ABB RAPID module: RobData.mod

MODULE RobData
    PERS num nHeigh:=-2.5;
	CONST speeddata vSlow:=[10,5,5,1000];
	CONST robtarget pTemp:=[[36.61,-311.94,82.16],[3.72224E-05,-1,-4.64438E-05,2.60135E-05],[-1,-1,-1,0],[9E+09,9E+09,9E+09,9E+09,9E+09,9E+09]];
	CONST speeddata vSlowA:=[2,5,5,1000];
    PERS robtarget phome1:=[[-40.4314,-257.966,143.781],[4.99019E-05,-0.667497,0.744613,6.30517E-05],[-2,-1,-1,0],[9E+09,9E+09,9E+09,9E+09,9E+09,9E+09]];
    PERS robtarget phome:=[[-122.06,-373,117.55],[3.74264E-05,-0.659781,0.751458,3.53401E-05],[-2,-1,-1,0],[9E+09,9E+09,9E+09,9E+09,9E+09,9E+09]];
	PERS robtarget pPickWait:=[[-121.80,-372.62,142.89],[4.48442E-05,-0.659779,0.751459,4.07139E-05],[-2,-1,-1,0],[9E+09,9E+09,9E+09,9E+09,9E+09,9E+09]];
    PERS robtarget pTCPCalib:=[[38.86,-315.26,82.1995],[4.51814E-05,-6.4519E-06,-1,-4.06358E-05],[-1,-1,-1,0],[9E+09,9E+09,9E+09,9E+09,9E+09,9E+09]];

    PERS robtarget pPass1:=[[200.53,-307.58,242.84],[0.299987,0.731588,0.298484,-0.534504],[-1,-1,-1,0],[9E+09,9E+09,9E+09,9E+09,9E+09,9E+09]];
    PERS robtarget pPass2:=[[887.04,835.36,1127.78],[0.0262232,0.74592,-0.665204,-0.0204732],[0,-2,-1,0],[9E+09,9E+09,9E+09,9E+09,9E+09,9E+09]];
    PERS robtarget pAssembly:=[[0,0,118],[0,-1,0,0],[-1,0,-1,0],[9E+09,9E+09,9E+09,9E+09,9E+09,9E+09]];
	PERS robtarget pAssem:=[[354.53,109.44,1307.28],[0.522631,-0.494622,0.5135,0.467465],[0,-1,-1,0],[9E+09,9E+09,9E+09,9E+09,9E+09,9E+09]];
    PERS robtarget pAssBase:=[[225.06,-308.31,118.65],[0.0102026,-0.99364,-0.111268,-0.0139692],[-1,0,-1,0],[9E+09,9E+09,9E+09,9E+09,9E+09,9E+09]];
    PERS robtarget pCali2Temp:=[[221.471,-305.943,140.42],[3.87751E-06,0.113366,-0.993553,-6.74824E-05],[-1,0,-1,0],[9E+09,9E+09,9E+09,9E+09,9E+09,9E+09]];
    VAR robtarget pActPos:=[[752.23,113.39,1307.28],[0.522626,-0.494634,0.513503,0.467454],[0,-2,0,0],[9E+09,9E+09,9E+09,9E+09,9E+09,9E+09]];
    PERS tooldata tGripper:=[TRUE,[[0,0,108],[0,0,0,-1]],[1,[0,0,0.001],[1,0,0,0],0,0,0]];
    PERS tooldata tcp1:=[TRUE,[[-134.881,-2.6021,210.993],[0.472574,-0.509839,-0.505206,0.511376]],[0.001,[0,0,0.001],[1,0,0,0],0,0,0]];
    PERS tooldata tcp2:=[TRUE,[[-134.881,-2.6021,210.993],[0.472574,-0.509839,-0.505206,0.511376]],[0.001,[0,0,0.001],[1,0,0,0],0,0,0]];
    PERS tooldata tCurTool:=[TRUE,[[0.0931091,-0.0380325,108],[0.998678,-1.1568E-12,-2.18595E-12,-0.0514118]],[1,[0,0,0.001],[1,0,0,0],0,0,0]];
    PERS wobjdata AssFrame:=[FALSE,TRUE,"",[[227.126,-306.421,7],[0.49417,0,0,-0.869366]],[[0,0,0],[1,0,0,0]]];
    PERS pose posRel:=[[27.92,-310.994,91.58],[3.54519E-05,-0.70071,-0.713446,3.18553E-08]];
    !the position of insert action
    PERS robtarget pccd2Calib{9}:=[[[221.89,-312.11,153.7],[6.08179E-05,-0.667482,0.744626,7.205E-05],[-1,0,0,0],[9E+09,9E+09,9E+09,9E+09,9E+09,9E+09]],[[221.89,-308.11,153.7],[6.08179E-05,-0.667482,0.744626,7.205E-05],[-1,0,0,0],[9E+09,9E+09,9E+09,9E+09,9E+09,9E+09]],[[221.89,-304.11,153.7],[6.08179E-05,-0.667482,0.744626,7.205E-05],[-1,0,0,0],[9E+09,9E+09,9E+09,9E+09,9E+09,9E+09]],[[225.89,-312.11,153.7],[6.08179E-05,-0.667482,0.744626,7.205E-05],[-1,0,0,0],[9E+09,9E+09,9E+09,9E+09,9E+09,9E+09]],[[225.89,-308.11,153.7],[6.08179E-05,-0.667482,0.744626,7.205E-05],[-1,0,0,0],[9E+09,9E+09,9E+09,9E+09,9E+09,9E+09]],[[225.89,-304.11,153.7],[6.08179E-05,-0.667482,0.744626,7.205E-05],[-1,0,0,0],[9E+09,9E+09,9E+09,9E+09,9E+09,9E+09]],[[229.89,-312.11,153.7],[6.08179E-05,-0.667482,0.744626,7.205E-05],[-1,0,0,0],[9E+09,9E+09,9E+09,9E+09,9E+09,9E+09]],[[229.89,-308.11,153.7],[6.08179E-05,-0.667482,0.744626,7.205E-05],[-1,0,0,0],[9E+09,9E+09,9E+09,9E+09,9E+09,9E+09]],[[229.89,-304.11,153.7],[6.08179E-05,-0.667482,0.744626,7.205E-05],[-1,0,0,0],[9E+09,9E+09,9E+09,9E+09,9E+09,9E+09]]];
    PERS string sCCD;
    PERS string sFirstStr;
    PERS string sSecondStr;
    PERS num Zangle:=-96.2517;
    PERS num Yangle:=0.00908074;
    PERS num Xangle:=179.998;
    VAR string CCD1X{9}:=["","","","","","","","",""];
    VAR string CCD1Y{9}:=["","","","","","","","",""];
    VAR string CCD2X{9}:=["","","","","","","","",""];
    VAR string CCD2Y{9}:=["","","","","","","","",""];
    PERS NUM ARRAY{9}:=[3,6,9,8,5,2,1,4,7];
    VAR string sCCD1;
    VAR string sCCD3;
    PERS num nanglex:=0;
    PERS num nangley:=0;
    !CCD 1 data for pick the Buttun
    PERS num X1:=27.92;
    PERS num Y1:=-310.994;
    PERS num nAngle1:=-88.968;
    !CCD2 data for gasket
    PERS num X2:=227.126;
    PERS num Y2:=-306.421;
    PERS num nAngle2:=-30.77;
    !CCD3 data for cable;
    PERS num X3:=0;
    PERS num Y3:=0;
    PERS num nAngle3:=0;
    PERS num X4:=35.818;
    PERS num Y4:=-312.359;
    PERS num nAngle4:=1.27;
    !the data from computer to modify the robot position

    !CCD3 data for cable;
    PERS num noffsX:=0.01;
    PERS num noffsY:=-0.28;
    PERS num noffsAngle:=0;
    PERS num nAssX:=0;
    PERS num nAssY:=0;
    PERS num nAssz:=0;
    PERS num XC:=0;
    PERS num YC:=0;
    PERS num nCCD:=0;
    PERS num nccd3offs:=0;
    PERS num nccd3offsx:=0;
    PERS num nTempX:=0;
    PERS num nTempY:=0;
    PERS num nTempZ:=0;
    PERS num nTAnglez:=0;
    PERS num nTAngley:=0;
    PERS num nTAnglex:=0;
    PERS num nPositionNo:=0;
    PERS num nHtemp:=0;
    !the insert speed of the robot
    PERS speeddata vAssembly:=[200,25,5000,1000];
    PERS num baseX2:=0;
    PERS num baseY2:=0;
    PERS bool bFull:=TRUE;
    PERS bool bWork:=FALSE;
    PERS bool bCalibration:=FALSE;
    PERS bool bInitall:=FALSE;
    PERS bool bEmptyDone:=FALSE;
    PERS bool SockGet:=TRUE;
    VAR intnum iSocketError:=0;
    VAR intnum iCalibration:=0;
    VAR intnum iInitall:=0;
    VAR intnum iEmptydone:=0;
    !CCD3 data for
    PERS num CCD1_X:=425.2;
    PERS num CCD1_Y:=-118.686;
    PERS num AngZ:=0;
    VAR socketdev temp_socket;
    PERS tooldata tGrip:=[TRUE,[[0,0,108],[1,0,0,0]],[2,[0,1,0],[1,0,0,0],0,0,0]];
    PERS tooldata tTCP:=[TRUE,[[0,0,120],[1,0,0,0]],[2,[0,1,0],[1,0,0,0],0,0,0]];
    PERS num n:=2;
    PERS num b:=3;
    PERS num nStrLength:=11;
    PERS num nfind:=42;
    PERS num nArray{9}:=[11,17,24,30,36,42,59,66,73];
    var num nArray1{9}:=[13,20,29,37,45,54,59,66,73];
    var num nArray2{3}:=[11,18,0];
    PERS pose nPoseAss:=[[0,0,0],[1,0,0,0]];
    PERS pos nPOSCCD1{9}:=[[23.9498,-313.292,91.5811],[23.9504,-311.091,91.5806],[23.9503,-308.89,91.5797],[27.9502,-313.292,91.5805],[27.9498,-311.09,91.5799],[27.9502,-308.889,91.5795],[31.95,-313.291,91.5805],[31.9497,-311.09,91.5799],[31.9495,-308.889,91.58]];
    PERS pos nPOSCCD2{9}:=[[223.894,-306.117,153.693],[225.893,-306.115,153.691],[227.893,-306.115,153.693],[227.893,-308.117,153.693],[225.893,-308.116,153.693],[223.895,-308.118,153.694],[223.893,-310.115,153.692],[225.892,-310.115,153.691],[227.892,-310.115,153.692]];
    PERS String SocketStr:="";
    PERS String SendStr:="";
    PERS String sFrame:="world";
    CONST robtarget p300:=[[35.94,-312.18,78.08],[0.0367958,-0.00985026,-0.999273,0.00150693],[-1,-1,-1,0],[9E+09,9E+09,9E+09,9E+09,9E+09,9E+09]];
    PERS robtarget pccd2Calib_T{9}:=[[[223.89,-310.11,153.7],[6.08179E-05,-0.667482,0.744626,7.205E-05],[-1,0,0,0],[9E+09,9E+09,9E+09,9E+09,9E+09,9E+09]],[[223.89,-308.11,153.7],[6.08179E-05,-0.667482,0.744626,7.205E-05],[-1,0,0,0],[9E+09,9E+09,9E+09,9E+09,9E+09,9E+09]],[[223.89,-306.11,153.7],[6.08179E-05,-0.667482,0.744626,7.205E-05],[-1,0,0,0],[9E+09,9E+09,9E+09,9E+09,9E+09,9E+09]],[[225.89,-310.11,153.7],[6.08179E-05,-0.667482,0.744626,7.205E-05],[-1,0,0,0],[9E+09,9E+09,9E+09,9E+09,9E+09,9E+09]],[[225.89,-308.11,153.7],[6.08179E-05,-0.667482,0.744626,7.205E-05],[-1,0,0,0],[9E+09,9E+09,9E+09,9E+09,9E+09,9E+09]],[[225.89,-306.11,153.7],[6.08179E-05,-0.667482,0.744626,7.205E-05],[-1,0,0,0],[9E+09,9E+09,9E+09,9E+09,9E+09,9E+09]],[[227.89,-310.11,153.7],[6.08179E-05,-0.667482,0.744626,7.205E-05],[-1,0,0,0],[9E+09,9E+09,9E+09,9E+09,9E+09,9E+09]],[[227.89,-308.11,153.7],[6.08179E-05,-0.667482,0.744626,7.205E-05],[-1,0,0,0],[9E+09,9E+09,9E+09,9E+09,9E+09,9E+09]],[[227.89,-306.11,153.7],[6.08179E-05,-0.667482,0.744626,7.205E-05],[-1,0,0,0],[9E+09,9E+09,9E+09,9E+09,9E+09,9E+09]]];
    VAR intnum intDoor:=0;
    PERS wobjdata AssFrame1:=[FALSE,TRUE,"",[[227.179,-306.738,7],[0.964165,0,0,-0.265304]],[[0,0,0],[1,0,0,0]]];
ENDMODULE
